// TIA Portal V20 export
DATA_BLOCK "DB_Digital_Outputs"   // DB3
{ S7_Optimized_Access := 'TRUE' }
// stored: AutoNumber false, MemoryReserve 100
   VAR
      Blink_Button_Light : Bool;
      Turn_On_Button_Light : Bool;
      Light_Fail_Test : Bool;
      Light_Approve_Test : Bool;
      Digital_Output_3 : Bool;
   END_VAR
BEGIN
END_DATA_BLOCK
